(* Schneider Machine Expert - Basic project Project_M221_ModbusRTU_Master, file version 2.8.0.0 *)
(* ProjectInformations: Name=New project *)

HARDWARE
  Cpu 0: TM221ME16T/G
  ModuleExtensionObject 0: TM3SAF5R/G
  EthernetConfiguration: NetworkName=M221, IpAllocationMode=FixedAddress, IpAddress=192.168.5.84, SubnetMask=255.255.255.0
  SerialLineConfiguration: Baud=Baud115200, Parity=ParityEven, DataBits=DataBits8, StopBits=StopBits1, PhysicalMedium=PhysicalMediumRs485, TransmissionMode=TransmissionModeModbusRtu, SlaveId=1, Addressing=MasterAddressing
  MastTask: UsePeriodScanMode=true, PeriodScan=1
  FastTask: Period=255
  CpuBehavior: StartingMode=StartAsPreviousState, AutoSaveRamOnEeprom=true, WatchdogPeriod=250

SYMBOLS  (address, symbol, comment, settings)
  %M0       HMI_SW_ADD1
  %M1       HMI_SW_RESET
  %M2       HMI_LP_INSETPOINT
  %M10      READVAR_MODE03_EXEXUTE
  %M11      READVAR_MODE03_ABORT
  %M12      READVAR_MODE03_DONE
  %M13      READVAR_MODE03_BUSY
  %M14      READVAR_MODE03_ABORTED
  %M15      READVAR_MODE03_ERROR
  %M20      WRITEVAR_MODE10_EXECUTE
  %M21      WRITEVAR_MODE10_ABORT
  %M22      WRITEVAR_MODE10_DONE
  %M23      WRITEVAR_MODE10_BUSY
  %M24      WRITEVAR_MODE10_ABORTED
  %M25      WRITEVAR_MODE10_ERROR
  %M30      READVAR_MODE02_EXECUTE
  %M31      READVAR_MODE02_ABORT
  %M32      READVAR_MODE02_DONE
  %M33      READVAR_MODE02_BUSY
  %M34      READVAR_MODE02_ABORTED
  %M35      READVAR_MODE02_ERROR
  %M40      WRITEVAR_MODE0F_EXECUTE
  %M41      WRITEVAR_MODE0F_ABORT
  %M42      WRITEVAR_MODE0F_DONE
  %M43      WRITEVAR_MODE0F_BUSY
  %M44      WRITEVAR_MODE0F_ABORTED
  %M45      WRITEVAR_MODE0F_ERROR
  %M50      READVAR_MODE01_EXECUTE
  %M51      READVAR_MODE01_ABORT
  %M52      READVAR_MODE01_DONE
  %M53      READVAR_MODE01_BUSY
  %M54      READVAR_MODE01_ABORTED
  %M55      READVAR_MODE01_ERROR
  %M60      WRITEVAR_MODE06_EXECUTE
  %M61      WRITEVAR_MODE06_ABORT
  %M62      WRITEVAR_MODE06_DONE
  %M63      WRITEVAR_MODE06_BUSY
  %M64      WRITEVAR_MODE06_ABORTED
  %M65      WRITEVAR_MODE06_ERROR
  %M70      WRITEVAR_MODE05_EXECUTE
  %M71      WRITEVAR_MODE05_ABORT
  %M72      WRITEVAR_MODE05_DONE
  %M73      WRITEVAR_MODE05_BUSY
  %M74      WRITEVAR_MODE05_ABORTED
  %M75      WRITEVAR_MODE05_ERROR
  %M80      READVAR_MODE04_EXECUTE
  %M81      READVAR_MODE04_ABORT
  %M82      READVAR_MODE04_DONE
  %M83      READVAR_MODE04_BUSY
  %M84      READVAR_MODE04_ABORTED
  %M85      READVAR_MODE04_ERROR
  %M100       "VALID"
  %M101       "ERRORSTOP"
  %M102       "DISABLED"
  %M103       "STOPPING"
  %M104       "STANDSTILL"
  %M105       "CONTMOTION"
  %M106       "ERROR"
  %M107       "DONE"
  %M108       "BUSY"
  %M109       "ERROR"
  %M500     DUMMY
  %S12      SB_RUNMODE  "The controller is running"
  %MW0      RTU_REGISTER_0
  %MW1      ISTEP
  %MW2      RTU_REGISTER_2
  %MW3      OKCOUNT
  %MW4      RTU_REGISTER_4
  %MW5      RTU_REGISTER_5
  %MW6      RTU_REGISTER_6
  %MW7      RTU_REGISTER_7
  %MW8      RTU_REGISTER_8
  %MW9      RTU_REGISTER_9
  %MW10     RTU_REGISTER_10
  %MW11     RTU_REGISTER_11
  %MW12     RTU_REGISTER_12
  %MW13     RTU_REGISTER_13
  %MW14     RTU_REGISTER_14
  %MW100    MULTIREGISTER_0
  %MW101    MULTIREGISTER_1
  %MW102    MULTIREGISTER_2
  %MW400    READ_VAR1_BUFFER
  %MW402    WRITE_VAR1_BUFFER
  %MW404    READ_VAR2_BUFFER
  %MW410    READ_VAR0_BUFFER0
  %MW411    READ_VAR0_BUFFER1
  %MW412    READ_VAR0_BUFFER2
  %MW413    READ_VAR0_BUFFER3
  %MW414    READ_VAR0_BUFFER4
  %MW415    READ_VAR0_BUFFER5
  %MW416    READ_VAR0_BUFFER6
  %MW417    READ_VAR0_BUFFER7
  %MW418    READ_VAR0_BUFFER8
  %MW419    READ_VAR0_BUFFER9
  %MW420    READ_VAR3_BUFFER0
  %MW421    READ_VAR3_BUFFER1
  %MW422    READ_VAR3_BUFFER2
  %MW423    READ_VAR3_BUFFER3
  %MW424    READ_VAR3_BUFFER4
  %MW425    READ_VAR3_BUFFER5
  %MW426    READ_VAR3_BUFFER6
  %MW427    READ_VAR3_BUFFER7
  %MW428    READ_VAR3_BUFFER8
  %MW429    READ_VAR3_BUFFER9
  %MW430    WRITE_VAR0_BUFFER0
  %MW431    WRITE_VAR0_BUFFER1
  %MW432    WRITE_VAR0_BUFFER2
  %MW433    WRITE_VAR0_BUFFER3
  %MW434    WRITE_VAR0_BUFFER4
  %MW435    WRITE_VAR0_BUFFER5
  %MW436    WRITE_VAR0_BUFFER6
  %MW437    WRITE_VAR0_BUFFER7
  %MW438    WRITE_VAR0_BUFFER8
  %MW439    WRITE_VAR0_BUFFER9
  %MW440    WRITE_VAR2_BUFFER0
  %MW441    WRITE_VAR3_BUFFER0
  %READ_VAR0 RTU_ID1_READ400000_10  [Link(Value(FBComLinkParameterEnums=SerialLine1)), RemoteDeviceId(Value(int=1)), Timeout(Value(int=200)), ObjType(Value(FBComObjTypeParameterEnums=MW)), FirstObj(Value(int=0)), Quantity(Value(int=10)), IndexData(Value(int=410))]
  %READ_VAR1 RTU_ID1_READ000000_16  [Link(Value(FBComLinkParameterEnums=SerialLine1)), RemoteDeviceId(Value(int=1)), Timeout(Value(int=100)), ObjType(Value(FBComObjTypeParameterEnums=I)), FirstObj(Value(int=0)), Quantity(Value(int=16)), IndexData(Value(int=400))]
  %READ_VAR2 RTU_ID1_READ000001_16  [Link(Value(FBComLinkParameterEnums=SerialLine1)), RemoteDeviceId(Value(int=1)), Timeout(Value(int=100)), ObjType(Value(FBComObjTypeParameterEnums=Q)), FirstObj(Value(int=0)), Quantity(Value(int=16)), IndexData(Value(int=404))]
  %READ_VAR3 RTU_ID1_READ300000_10  [Link(Value(FBComLinkParameterEnums=SerialLine1)), RemoteDeviceId(Value(int=1)), Timeout(Value(int=100)), ObjType(Value(FBComObjTypeParameterEnums=IW)), FirstObj(Value(int=0)), Quantity(Value(int=10)), IndexData(Value(int=420))]
  %WRITE_VAR0 RTU_ID1_WRITE300000_10  [Link(Value(FBComLinkParameterEnums=SerialLine1)), RemoteDeviceId(Value(int=1)), Timeout(Value(int=100)), ObjType(Value(FBComObjTypeParameterEnums=MW)), FirstObj(Value(int=0)), Quantity(Value(int=10)), IndexData(Value(int=430))]
  %WRITE_VAR1 RTU_ID1_WRITE000000_16  [Link(Value(FBComLinkParameterEnums=SerialLine1)), RemoteDeviceId(Value(int=1)), Timeout(Value(int=100)), ObjType(Value(FBComObjTypeParameterEnums=Q)), FirstObj(Value(int=0)), Quantity(Value(int=16)), IndexData(Value(int=402))]
  %WRITE_VAR2 RTU_ID1_WRITE400000_1  [Link(Value(FBComLinkParameterEnums=SerialLine1)), RemoteDeviceId(Value(int=1)), Timeout(Value(int=100)), ObjType(Value(FBComObjTypeParameterEnums=SINGLE_REG)), FirstObj(Value(int=14)), Quantity(Value(int=1)), IndexData(Value(int=440))]
  %WRITE_VAR3 RTU_ID1_WRITE000000_1  [Link(Value(FBComLinkParameterEnums=SerialLine1)), RemoteDeviceId(Value(int=1)), Timeout(Value(int=100)), ObjType(Value(FBComObjTypeParameterEnums=SINGLE_COIL)), FirstObj(Value(int=0)), Quantity(Value(int=1)), IndexData(Value(int=441))]
  %QWM0     MODBUS_QWM0
  %QWM1     MODBUS_QWM1
  %QWM2     MODBUS_QWM2
  %QWM3     MODBUS_QWM3
  %QWM4     MODBUS_QWM4
  %QWM5     MODBUS_QWM5
  %QWM6     MODBUS_QWM6
  %QWM7     MODBUS_QWM7
  %QWM8     MODBUS_QWM8
  %QWM9     MODBUS_QWM9
  %QWM10    MODBUS_QWM10
  %QWM11    MODBUS_QWM11
  %QWM12    MODBUS_QWM12
  %QWM13    MODBUS_QWM13
  %QWM14    MODBUS_QWM14
  %QWM15    MODBUS_QWM15
  %QWM16    MODBUS_QWM16
  %QWM17    MODBUS_QWM17
  %QWM18    MODBUS_QWM18
  %QWM19    MODBUS_QWM19
  %IWM0     MODBUS_IWM0
  %IWM1     MODBUS_IWM1
  %IWM2     MODBUS_IWM2
  %IWM3     MODBUS_IWM3
  %IWM4     MODBUS_IWM4
  %IWM5     MODBUS_IWM5
  %IWM6     MODBUS_IWM6
  %IWM7     MODBUS_IWM7
  %IWM8     MODBUS_IWM8
  %IWM9     MODBUS_IWM9
  %IWM10    MODBUS_IWM10
  %IWM11    MODBUS_IWM11
  %IWM12    MODBUS_IWM12
  %IWM13    MODBUS_IWM13
  %IWM14    MODBUS_IWM14
  %IWM15    MODBUS_IWM15
  %IWM16    MODBUS_IWM16
  %IWM17    MODBUS_IWM17
  %IWM18    MODBUS_IWM18
  %IWM19    MODBUS_IWM19
  %I1.8       "Reserved"
  %I1.13      "Reserved"
  %Q1.3       "Reserved"

POU Pou01_System
  (* SectionNumber=1 *)

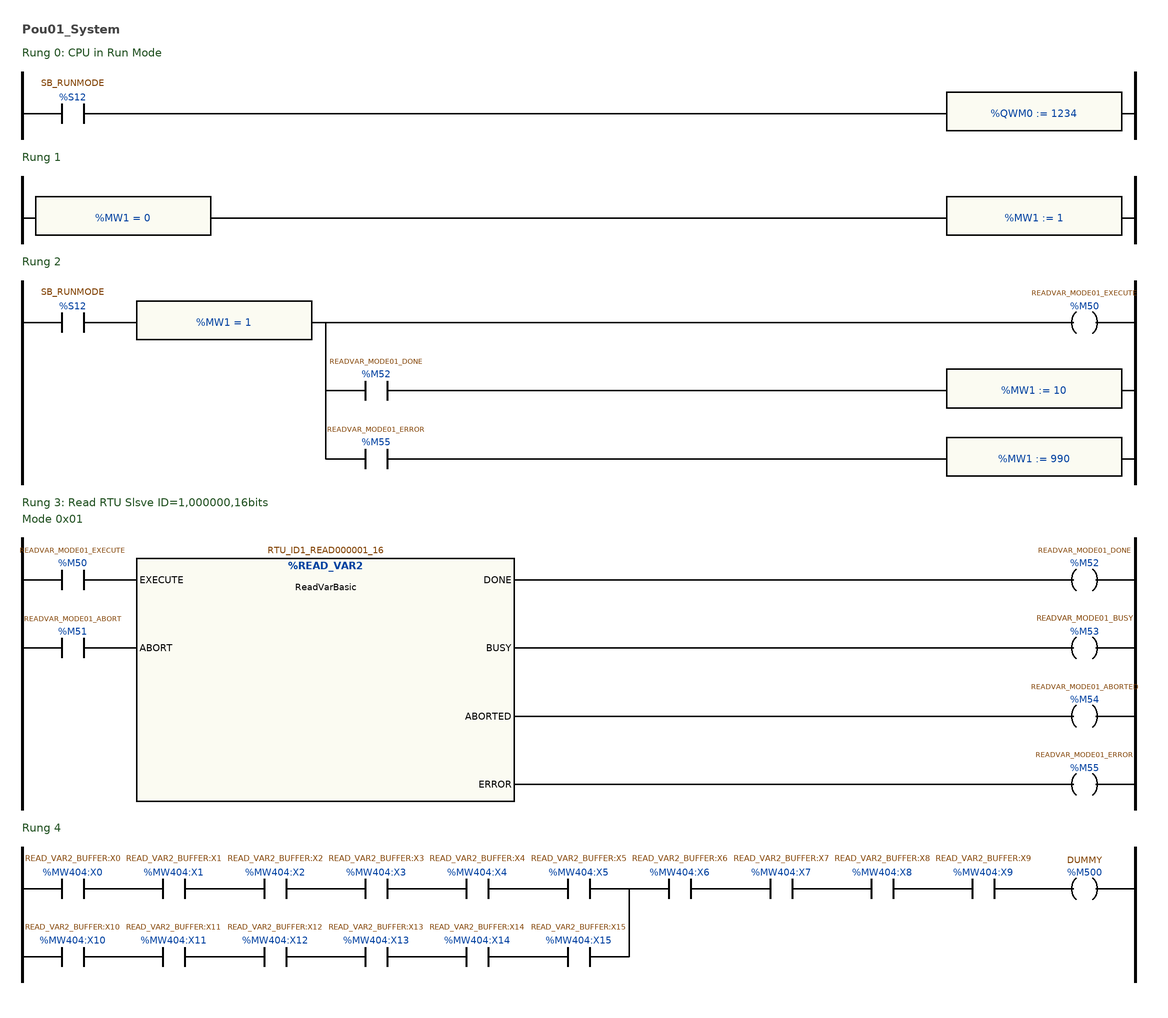

// Rung 0: CPU in Run Mode
  LD %S12                 (* SB_RUNMODE *)
  [ %QWM0 := 1234 ]       (* MODBUS_QWM0 *)
  // as ST:
  //   IF SB_RUNMODE THEN MODBUS_QWM0 := 1234; END_IF;

// Rung 1
  LD [ %MW1 = 0 ]         (* ISTEP *)
  [ %MW1 := 1 ]           (* ISTEP *)
  // as ST:
  //   IF ISTEP = 0 THEN ISTEP := 1; END_IF;

// Rung 2
  LD %S12                 (* SB_RUNMODE *)
  AND [ %MW1 = 1 ]        (* ISTEP *)
  MPS
  ST %M50                 (* READVAR_MODE01_EXECUTE *)
  MRD
  AND %M52                (* READVAR_MODE01_DONE *)
  [ %MW1 := 10 ]          (* ISTEP *)
  MPP
  AND %M55                (* READVAR_MODE01_ERROR *)
  [ %MW1 := 990 ]         (* ISTEP *)
  // as ST:
  //   READVAR_MODE01_EXECUTE := SB_RUNMODE AND ISTEP = 1;
  //   _t1 := SB_RUNMODE AND ISTEP = 1;
  //   IF SB_RUNMODE AND ISTEP = 1 AND READVAR_MODE01_DONE THEN ISTEP := 10; END_IF;
  //   IF _t1 AND READVAR_MODE01_ERROR THEN ISTEP := 990; END_IF;

// Rung 3: Read RTU Slsve ID=1,000000,16bits
// Mode 0x01
  BLK %READ_VAR2
  LD %M50                 (* READVAR_MODE01_EXECUTE *)
  EXECUTE
  LD %M51                 (* READVAR_MODE01_ABORT *)
  ABORT
  OUT_BLK
  LD DONE
  ST %M52                 (* READVAR_MODE01_DONE *)
  LD BUSY
  ST %M53                 (* READVAR_MODE01_BUSY *)
  LD ABORTED
  ST %M54                 (* READVAR_MODE01_ABORTED *)
  LD ERROR
  ST %M55                 (* READVAR_MODE01_ERROR *)
  END_BLK
  // as ST:
  //   %READ_VAR2(EXECUTE := READVAR_MODE01_EXECUTE, ABORT := READVAR_MODE01_ABORT);
  //   READVAR_MODE01_DONE := %READ_VAR2.DONE;
  //   READVAR_MODE01_BUSY := %READ_VAR2.BUSY;
  //   READVAR_MODE01_ABORTED := %READ_VAR2.ABORTED;
  //   READVAR_MODE01_ERROR := %READ_VAR2.ERROR;

// Rung 4
  LD %MW404:X0            (* READ_VAR2_BUFFER *)
  AND %MW404:X1           (* READ_VAR2_BUFFER *)
  AND %MW404:X2           (* READ_VAR2_BUFFER *)
  AND %MW404:X3           (* READ_VAR2_BUFFER *)
  AND %MW404:X4           (* READ_VAR2_BUFFER *)
  AND %MW404:X5           (* READ_VAR2_BUFFER *)
  OR( %MW404:X10          (* READ_VAR2_BUFFER *)
  AND %MW404:X11          (* READ_VAR2_BUFFER *)
  AND %MW404:X12          (* READ_VAR2_BUFFER *)
  AND %MW404:X13          (* READ_VAR2_BUFFER *)
  AND %MW404:X14          (* READ_VAR2_BUFFER *)
  AND %MW404:X15          (* READ_VAR2_BUFFER *)
  )
  AND %MW404:X6           (* READ_VAR2_BUFFER *)
  AND %MW404:X7           (* READ_VAR2_BUFFER *)
  AND %MW404:X8           (* READ_VAR2_BUFFER *)
  AND %MW404:X9           (* READ_VAR2_BUFFER *)
  ST %M500                (* DUMMY *)
  // as ST:
  //   DUMMY := (READ_VAR2_BUFFER:X0 AND READ_VAR2_BUFFER:X1 AND READ_VAR2_BUFFER:X2 AND READ_VAR2_BUFFER:X3 AND READ_VAR2_BUFFER:X4 AND READ_VAR2_BUFFER:X5 OR READ_VAR2_BUFFER:X10 AND READ_VAR2_BUFFER:X11 AND READ_VAR2_BUFFER:X12 AND READ_VAR2_BUFFER:X13 AND READ_VAR2_BUFFER:X14 AND READ_VAR2_BUFFER:X15) AND READ_VAR2_BUFFER:X6 AND READ_VAR2_BUFFER:X7 AND READ_VAR2_BUFFER:X8 AND READ_VAR2_BUFFER:X9;

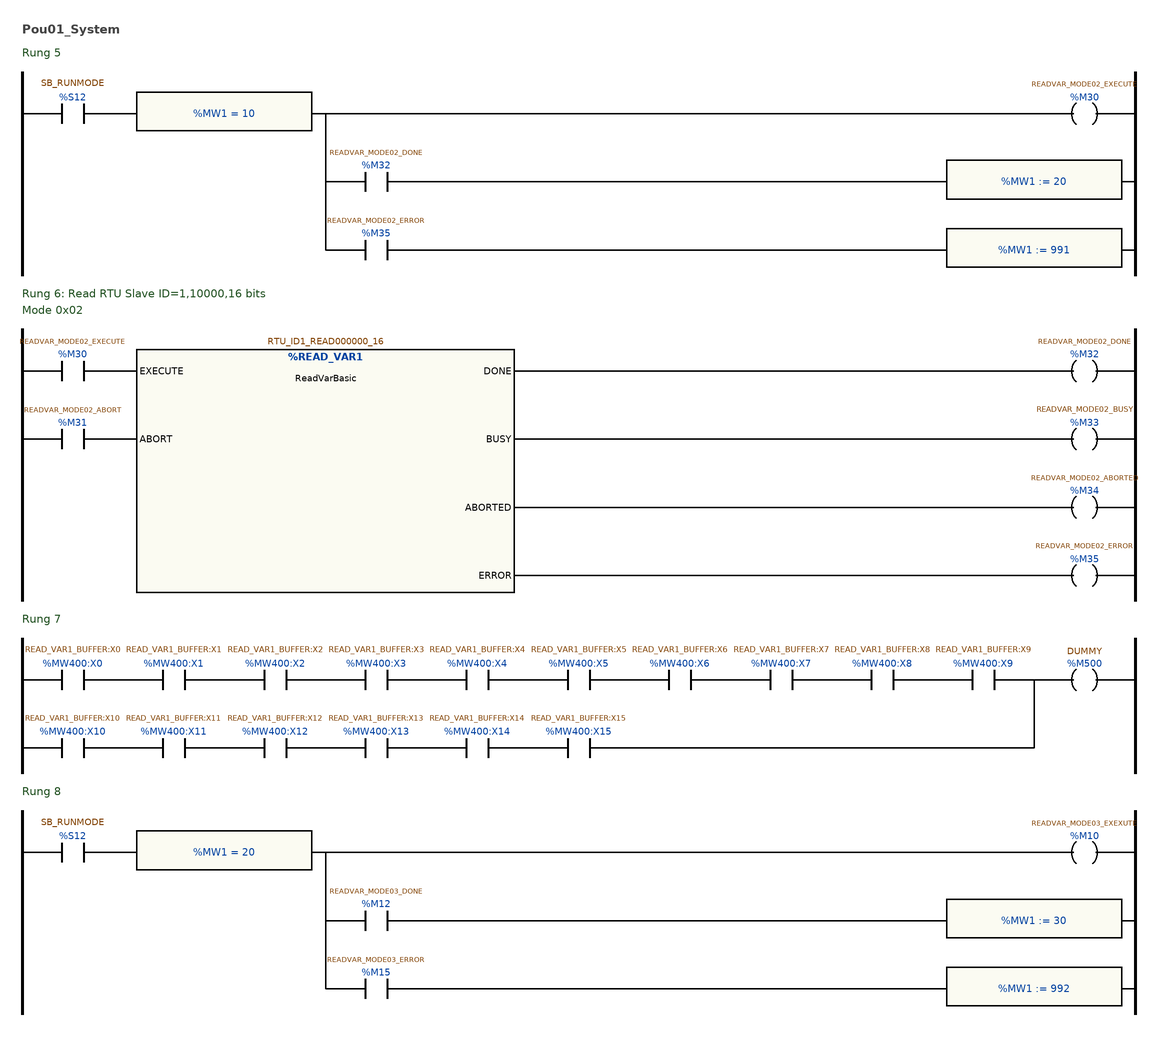

// Rung 5
  LD %S12                 (* SB_RUNMODE *)
  AND [ %MW1 = 10 ]       (* ISTEP *)
  MPS
  ST %M30                 (* READVAR_MODE02_EXECUTE *)
  MRD
  AND %M32                (* READVAR_MODE02_DONE *)
  [ %MW1 := 20 ]          (* ISTEP *)
  MPP
  AND %M35                (* READVAR_MODE02_ERROR *)
  [ %MW1 := 991 ]         (* ISTEP *)
  // as ST:
  //   READVAR_MODE02_EXECUTE := SB_RUNMODE AND ISTEP = 10;
  //   _t1 := SB_RUNMODE AND ISTEP = 10;
  //   IF SB_RUNMODE AND ISTEP = 10 AND READVAR_MODE02_DONE THEN ISTEP := 20; END_IF;
  //   IF _t1 AND READVAR_MODE02_ERROR THEN ISTEP := 991; END_IF;

// Rung 6: Read RTU Slave ID=1,10000,16 bits
// Mode 0x02
  BLK %READ_VAR1
  LD %M30                 (* READVAR_MODE02_EXECUTE *)
  EXECUTE
  LD %M31                 (* READVAR_MODE02_ABORT *)
  ABORT
  OUT_BLK
  LD DONE
  ST %M32                 (* READVAR_MODE02_DONE *)
  LD BUSY
  ST %M33                 (* READVAR_MODE02_BUSY *)
  LD ABORTED
  ST %M34                 (* READVAR_MODE02_ABORTED *)
  LD ERROR
  ST %M35                 (* READVAR_MODE02_ERROR *)
  END_BLK
  // as ST:
  //   %READ_VAR1(EXECUTE := READVAR_MODE02_EXECUTE, ABORT := READVAR_MODE02_ABORT);
  //   READVAR_MODE02_DONE := %READ_VAR1.DONE;
  //   READVAR_MODE02_BUSY := %READ_VAR1.BUSY;
  //   READVAR_MODE02_ABORTED := %READ_VAR1.ABORTED;
  //   READVAR_MODE02_ERROR := %READ_VAR1.ERROR;

// Rung 7
  LD %MW400:X0            (* READ_VAR1_BUFFER *)
  AND %MW400:X1           (* READ_VAR1_BUFFER *)
  AND %MW400:X2           (* READ_VAR1_BUFFER *)
  AND %MW400:X3           (* READ_VAR1_BUFFER *)
  AND %MW400:X4           (* READ_VAR1_BUFFER *)
  AND %MW400:X5           (* READ_VAR1_BUFFER *)
  AND %MW400:X6           (* READ_VAR1_BUFFER *)
  AND %MW400:X7           (* READ_VAR1_BUFFER *)
  AND %MW400:X8           (* READ_VAR1_BUFFER *)
  AND %MW400:X9           (* READ_VAR1_BUFFER *)
  OR( %MW400:X10          (* READ_VAR1_BUFFER *)
  AND %MW400:X11          (* READ_VAR1_BUFFER *)
  AND %MW400:X12          (* READ_VAR1_BUFFER *)
  AND %MW400:X13          (* READ_VAR1_BUFFER *)
  AND %MW400:X14          (* READ_VAR1_BUFFER *)
  AND %MW400:X15          (* READ_VAR1_BUFFER *)
  )
  ST %M500                (* DUMMY *)
  // as ST:
  //   DUMMY := READ_VAR1_BUFFER:X0 AND READ_VAR1_BUFFER:X1 AND READ_VAR1_BUFFER:X2 AND READ_VAR1_BUFFER:X3 AND READ_VAR1_BUFFER:X4 AND READ_VAR1_BUFFER:X5 AND READ_VAR1_BUFFER:X6 AND READ_VAR1_BUFFER:X7 AND READ_VAR1_BUFFER:X8 AND READ_VAR1_BUFFER:X9 OR READ_VAR1_BUFFER:X10 AND READ_VAR1_BUFFER:X11 AND READ_VAR1_BUFFER:X12 AND READ_VAR1_BUFFER:X13 AND READ_VAR1_BUFFER:X14 AND READ_VAR1_BUFFER:X15;

// Rung 8
  LD %S12                 (* SB_RUNMODE *)
  AND [ %MW1 = 20 ]       (* ISTEP *)
  MPS
  ST %M10                 (* READVAR_MODE03_EXEXUTE *)
  MRD
  AND %M12                (* READVAR_MODE03_DONE *)
  [ %MW1 := 30 ]          (* ISTEP *)
  MPP
  AND %M15                (* READVAR_MODE03_ERROR *)
  [ %MW1 := 992 ]         (* ISTEP *)
  // as ST:
  //   READVAR_MODE03_EXEXUTE := SB_RUNMODE AND ISTEP = 20;
  //   _t1 := SB_RUNMODE AND ISTEP = 20;
  //   IF SB_RUNMODE AND ISTEP = 20 AND READVAR_MODE03_DONE THEN ISTEP := 30; END_IF;
  //   IF _t1 AND READVAR_MODE03_ERROR THEN ISTEP := 992; END_IF;

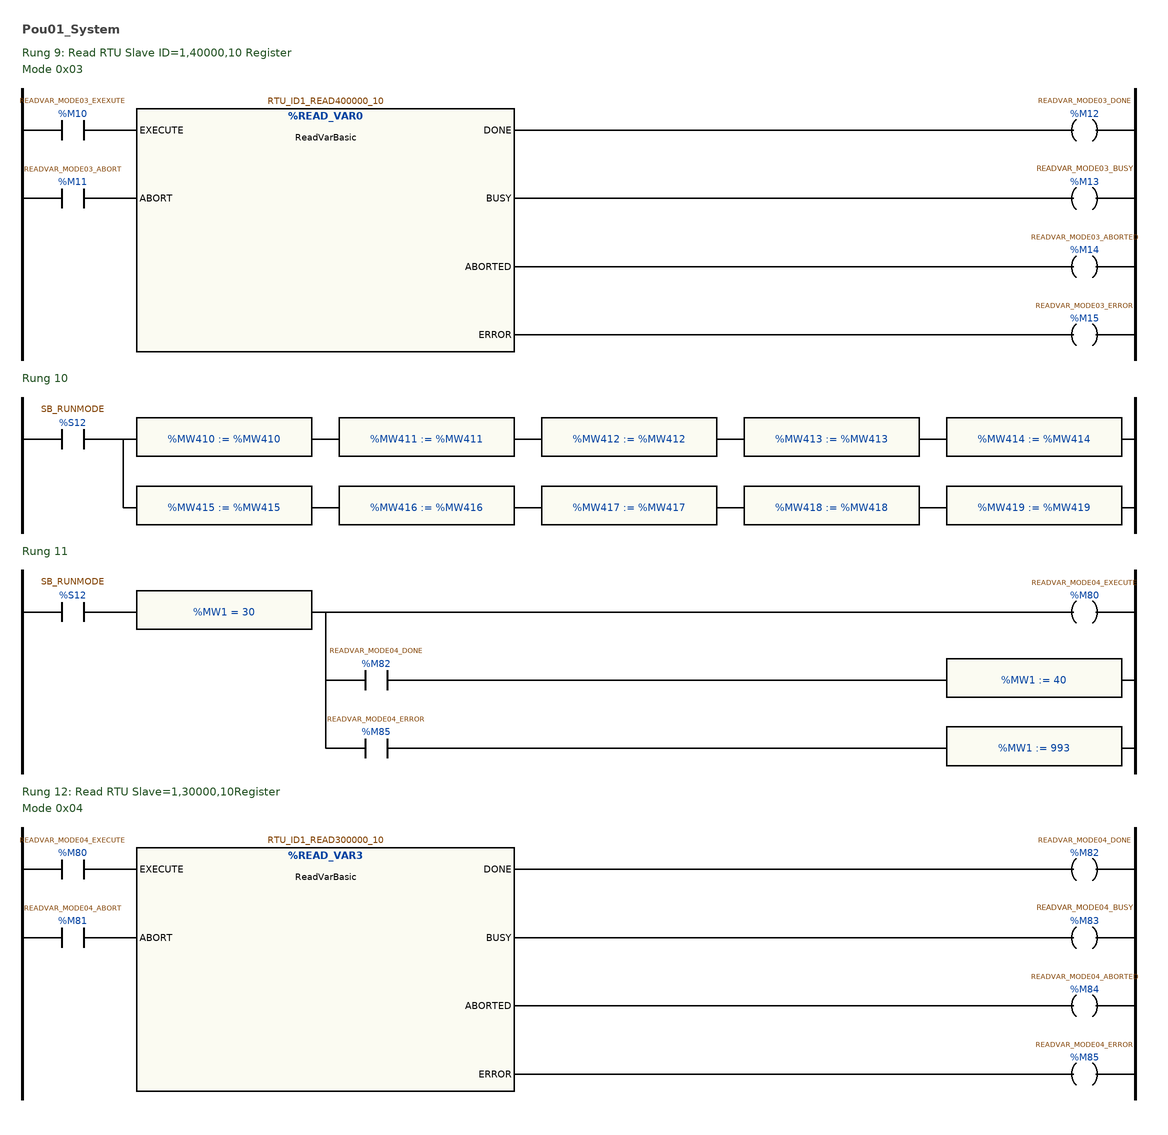

// Rung 9: Read RTU Slave ID=1,40000,10 Register
// Mode 0x03
  BLK %READ_VAR0
  LD %M10                 (* READVAR_MODE03_EXEXUTE *)
  EXECUTE
  LD %M11                 (* READVAR_MODE03_ABORT *)
  ABORT
  OUT_BLK
  LD DONE
  ST %M12                 (* READVAR_MODE03_DONE *)
  LD BUSY
  ST %M13                 (* READVAR_MODE03_BUSY *)
  LD ABORTED
  ST %M14                 (* READVAR_MODE03_ABORTED *)
  LD ERROR
  ST %M15                 (* READVAR_MODE03_ERROR *)
  END_BLK
  // as ST:
  //   %READ_VAR0(EXECUTE := READVAR_MODE03_EXEXUTE, ABORT := READVAR_MODE03_ABORT);
  //   READVAR_MODE03_DONE := %READ_VAR0.DONE;
  //   READVAR_MODE03_BUSY := %READ_VAR0.BUSY;
  //   READVAR_MODE03_ABORTED := %READ_VAR0.ABORTED;
  //   READVAR_MODE03_ERROR := %READ_VAR0.ERROR;

// Rung 10
  LD %S12                 (* SB_RUNMODE *)
  MPS
  OPER [ %MW410 := %MW410 ](* READ_VAR0_BUFFER0, READ_VAR0_BUFFER0 *)
  OPER [ %MW411 := %MW411 ](* READ_VAR0_BUFFER1, READ_VAR0_BUFFER1 *)
  OPER [ %MW412 := %MW412 ](* READ_VAR0_BUFFER2, READ_VAR0_BUFFER2 *)
  OPER [ %MW413 := %MW413 ](* READ_VAR0_BUFFER3, READ_VAR0_BUFFER3 *)
  [ %MW414 := %MW414 ]    (* READ_VAR0_BUFFER4, READ_VAR0_BUFFER4 *)
  MPP
  OPER [ %MW415 := %MW415 ](* READ_VAR0_BUFFER5, READ_VAR0_BUFFER5 *)
  OPER [ %MW416 := %MW416 ](* READ_VAR0_BUFFER6, READ_VAR0_BUFFER6 *)
  OPER [ %MW417 := %MW417 ](* READ_VAR0_BUFFER7, READ_VAR0_BUFFER7 *)
  OPER [ %MW418 := %MW418 ](* READ_VAR0_BUFFER8, READ_VAR0_BUFFER8 *)
  [ %MW419 := %MW419 ]    (* READ_VAR0_BUFFER9, READ_VAR0_BUFFER9 *)
  // as ST:
  //   IF SB_RUNMODE THEN READ_VAR0_BUFFER0 := READ_VAR0_BUFFER0; END_IF;
  //   IF SB_RUNMODE THEN READ_VAR0_BUFFER1 := READ_VAR0_BUFFER1; END_IF;
  //   IF SB_RUNMODE THEN READ_VAR0_BUFFER2 := READ_VAR0_BUFFER2; END_IF;
  //   IF SB_RUNMODE THEN READ_VAR0_BUFFER3 := READ_VAR0_BUFFER3; END_IF;
  //   IF SB_RUNMODE THEN READ_VAR0_BUFFER4 := READ_VAR0_BUFFER4; END_IF;
  //   IF SB_RUNMODE THEN READ_VAR0_BUFFER5 := READ_VAR0_BUFFER5; END_IF;
  //   IF SB_RUNMODE THEN READ_VAR0_BUFFER6 := READ_VAR0_BUFFER6; END_IF;
  //   IF SB_RUNMODE THEN READ_VAR0_BUFFER7 := READ_VAR0_BUFFER7; END_IF;
  //   IF SB_RUNMODE THEN READ_VAR0_BUFFER8 := READ_VAR0_BUFFER8; END_IF;
  //   IF SB_RUNMODE THEN READ_VAR0_BUFFER9 := READ_VAR0_BUFFER9; END_IF;

// Rung 11
  LD %S12                 (* SB_RUNMODE *)
  AND [ %MW1 = 30 ]       (* ISTEP *)
  MPS
  ST %M80                 (* READVAR_MODE04_EXECUTE *)
  MRD
  AND %M82                (* READVAR_MODE04_DONE *)
  [ %MW1 := 40 ]          (* ISTEP *)
  MPP
  AND %M85                (* READVAR_MODE04_ERROR *)
  [ %MW1 := 993 ]         (* ISTEP *)
  // as ST:
  //   READVAR_MODE04_EXECUTE := SB_RUNMODE AND ISTEP = 30;
  //   _t1 := SB_RUNMODE AND ISTEP = 30;
  //   IF SB_RUNMODE AND ISTEP = 30 AND READVAR_MODE04_DONE THEN ISTEP := 40; END_IF;
  //   IF _t1 AND READVAR_MODE04_ERROR THEN ISTEP := 993; END_IF;

// Rung 12: Read RTU Slave=1,30000,10Register
// Mode 0x04
  BLK %READ_VAR3
  LD %M80                 (* READVAR_MODE04_EXECUTE *)
  EXECUTE
  LD %M81                 (* READVAR_MODE04_ABORT *)
  ABORT
  OUT_BLK
  LD DONE
  ST %M82                 (* READVAR_MODE04_DONE *)
  LD BUSY
  ST %M83                 (* READVAR_MODE04_BUSY *)
  LD ABORTED
  ST %M84                 (* READVAR_MODE04_ABORTED *)
  LD ERROR
  ST %M85                 (* READVAR_MODE04_ERROR *)
  END_BLK
  // as ST:
  //   %READ_VAR3(EXECUTE := READVAR_MODE04_EXECUTE, ABORT := READVAR_MODE04_ABORT);
  //   READVAR_MODE04_DONE := %READ_VAR3.DONE;
  //   READVAR_MODE04_BUSY := %READ_VAR3.BUSY;
  //   READVAR_MODE04_ABORTED := %READ_VAR3.ABORTED;
  //   READVAR_MODE04_ERROR := %READ_VAR3.ERROR;

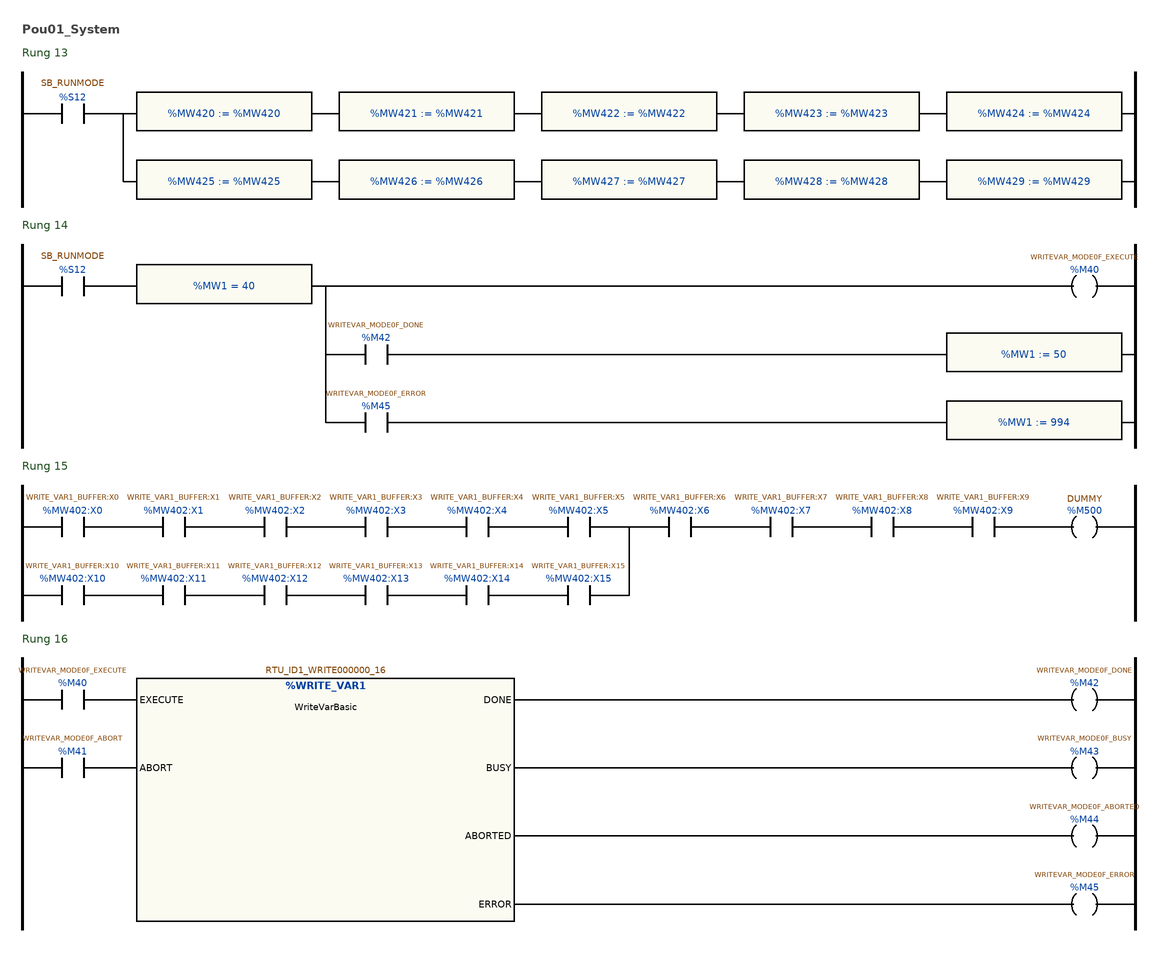

// Rung 13
  LD %S12                 (* SB_RUNMODE *)
  MPS
  OPER [ %MW420 := %MW420 ](* READ_VAR3_BUFFER0, READ_VAR3_BUFFER0 *)
  OPER [ %MW421 := %MW421 ](* READ_VAR3_BUFFER1, READ_VAR3_BUFFER1 *)
  OPER [ %MW422 := %MW422 ](* READ_VAR3_BUFFER2, READ_VAR3_BUFFER2 *)
  OPER [ %MW423 := %MW423 ](* READ_VAR3_BUFFER3, READ_VAR3_BUFFER3 *)
  [ %MW424 := %MW424 ]    (* READ_VAR3_BUFFER4, READ_VAR3_BUFFER4 *)
  MPP
  OPER [ %MW425 := %MW425 ](* READ_VAR3_BUFFER5, READ_VAR3_BUFFER5 *)
  OPER [ %MW426 := %MW426 ](* READ_VAR3_BUFFER6, READ_VAR3_BUFFER6 *)
  OPER [ %MW427 := %MW427 ](* READ_VAR3_BUFFER7, READ_VAR3_BUFFER7 *)
  OPER [ %MW428 := %MW428 ](* READ_VAR3_BUFFER8, READ_VAR3_BUFFER8 *)
  [ %MW429 := %MW429 ]    (* READ_VAR3_BUFFER9, READ_VAR3_BUFFER9 *)
  // as ST:
  //   IF SB_RUNMODE THEN READ_VAR3_BUFFER0 := READ_VAR3_BUFFER0; END_IF;
  //   IF SB_RUNMODE THEN READ_VAR3_BUFFER1 := READ_VAR3_BUFFER1; END_IF;
  //   IF SB_RUNMODE THEN READ_VAR3_BUFFER2 := READ_VAR3_BUFFER2; END_IF;
  //   IF SB_RUNMODE THEN READ_VAR3_BUFFER3 := READ_VAR3_BUFFER3; END_IF;
  //   IF SB_RUNMODE THEN READ_VAR3_BUFFER4 := READ_VAR3_BUFFER4; END_IF;
  //   IF SB_RUNMODE THEN READ_VAR3_BUFFER5 := READ_VAR3_BUFFER5; END_IF;
  //   IF SB_RUNMODE THEN READ_VAR3_BUFFER6 := READ_VAR3_BUFFER6; END_IF;
  //   IF SB_RUNMODE THEN READ_VAR3_BUFFER7 := READ_VAR3_BUFFER7; END_IF;
  //   IF SB_RUNMODE THEN READ_VAR3_BUFFER8 := READ_VAR3_BUFFER8; END_IF;
  //   IF SB_RUNMODE THEN READ_VAR3_BUFFER9 := READ_VAR3_BUFFER9; END_IF;

// Rung 14
  LD %S12                 (* SB_RUNMODE *)
  AND [ %MW1 = 40 ]       (* ISTEP *)
  MPS
  ST %M40                 (* WRITEVAR_MODE0F_EXECUTE *)
  MRD
  AND %M42                (* WRITEVAR_MODE0F_DONE *)
  [ %MW1 := 50 ]          (* ISTEP *)
  MPP
  AND %M45                (* WRITEVAR_MODE0F_ERROR *)
  [ %MW1 := 994 ]         (* ISTEP *)
  // as ST:
  //   WRITEVAR_MODE0F_EXECUTE := SB_RUNMODE AND ISTEP = 40;
  //   _t1 := SB_RUNMODE AND ISTEP = 40;
  //   IF SB_RUNMODE AND ISTEP = 40 AND WRITEVAR_MODE0F_DONE THEN ISTEP := 50; END_IF;
  //   IF _t1 AND WRITEVAR_MODE0F_ERROR THEN ISTEP := 994; END_IF;

// Rung 15
  LD %MW402:X0            (* WRITE_VAR1_BUFFER *)
  AND %MW402:X1           (* WRITE_VAR1_BUFFER *)
  AND %MW402:X2           (* WRITE_VAR1_BUFFER *)
  AND %MW402:X3           (* WRITE_VAR1_BUFFER *)
  AND %MW402:X4           (* WRITE_VAR1_BUFFER *)
  AND %MW402:X5           (* WRITE_VAR1_BUFFER *)
  OR( %MW402:X10          (* WRITE_VAR1_BUFFER *)
  AND %MW402:X11          (* WRITE_VAR1_BUFFER *)
  AND %MW402:X12          (* WRITE_VAR1_BUFFER *)
  AND %MW402:X13          (* WRITE_VAR1_BUFFER *)
  AND %MW402:X14          (* WRITE_VAR1_BUFFER *)
  AND %MW402:X15          (* WRITE_VAR1_BUFFER *)
  )
  AND %MW402:X6           (* WRITE_VAR1_BUFFER *)
  AND %MW402:X7           (* WRITE_VAR1_BUFFER *)
  AND %MW402:X8           (* WRITE_VAR1_BUFFER *)
  AND %MW402:X9           (* WRITE_VAR1_BUFFER *)
  ST %M500                (* DUMMY *)
  // as ST:
  //   DUMMY := (WRITE_VAR1_BUFFER:X0 AND WRITE_VAR1_BUFFER:X1 AND WRITE_VAR1_BUFFER:X2 AND WRITE_VAR1_BUFFER:X3 AND WRITE_VAR1_BUFFER:X4 AND WRITE_VAR1_BUFFER:X5 OR WRITE_VAR1_BUFFER:X10 AND WRITE_VAR1_BUFFER:X11 AND WRITE_VAR1_BUFFER:X12 AND WRITE_VAR1_BUFFER:X13 AND WRITE_VAR1_BUFFER:X14 AND WRITE_VAR1_BUFFER:X15) AND WRITE_VAR1_BUFFER:X6 AND WRITE_VAR1_BUFFER:X7 AND WRITE_VAR1_BUFFER:X8 AND WRITE_VAR1_BUFFER:X9;

// Rung 16
  BLK %WRITE_VAR1
  LD %M40                 (* WRITEVAR_MODE0F_EXECUTE *)
  EXECUTE
  LD %M41                 (* WRITEVAR_MODE0F_ABORT *)
  ABORT
  OUT_BLK
  LD DONE
  ST %M42                 (* WRITEVAR_MODE0F_DONE *)
  LD BUSY
  ST %M43                 (* WRITEVAR_MODE0F_BUSY *)
  LD ABORTED
  ST %M44                 (* WRITEVAR_MODE0F_ABORTED *)
  LD ERROR
  ST %M45                 (* WRITEVAR_MODE0F_ERROR *)
  END_BLK
  // as ST:
  //   %WRITE_VAR1(EXECUTE := WRITEVAR_MODE0F_EXECUTE, ABORT := WRITEVAR_MODE0F_ABORT);
  //   WRITEVAR_MODE0F_DONE := %WRITE_VAR1.DONE;
  //   WRITEVAR_MODE0F_BUSY := %WRITE_VAR1.BUSY;
  //   WRITEVAR_MODE0F_ABORTED := %WRITE_VAR1.ABORTED;
  //   WRITEVAR_MODE0F_ERROR := %WRITE_VAR1.ERROR;

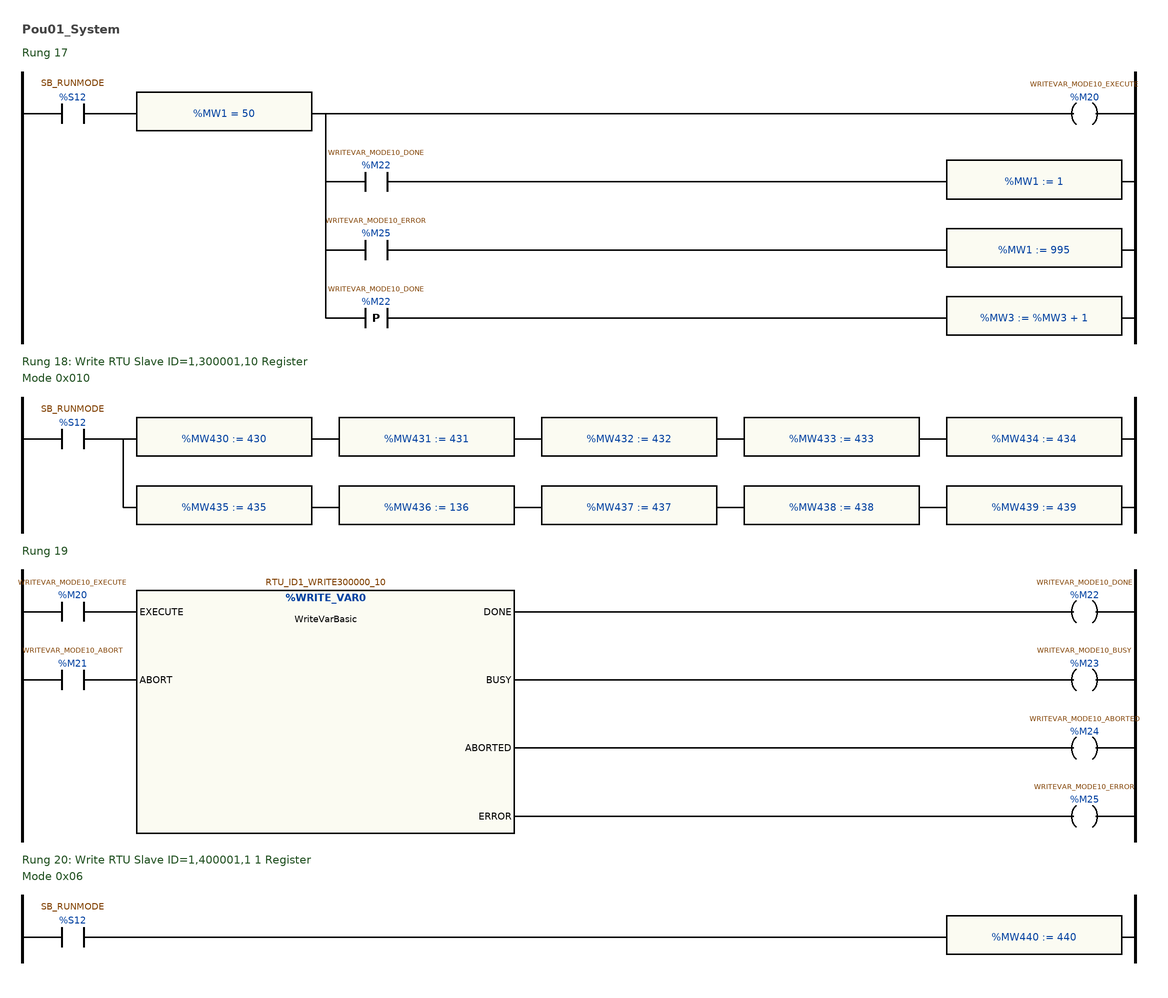

// Rung 17
  LD %S12                 (* SB_RUNMODE *)
  AND [ %MW1 = 50 ]       (* ISTEP *)
  MPS
  ST %M20                 (* WRITEVAR_MODE10_EXECUTE *)
  MRD
  AND %M22                (* WRITEVAR_MODE10_DONE *)
  [ %MW1 := 1 ]           (* ISTEP *)
  MRD
  AND %M25                (* WRITEVAR_MODE10_ERROR *)
  [ %MW1 := 995 ]         (* ISTEP *)
  MPP
  ANDR %M22               (* WRITEVAR_MODE10_DONE *)
  [ %MW3 := %MW3 + 1 ]    (* OKCOUNT, OKCOUNT *)
  // as ST:
  //   WRITEVAR_MODE10_EXECUTE := SB_RUNMODE AND ISTEP = 50;
  //   _t1 := SB_RUNMODE AND ISTEP = 50;
  //   IF SB_RUNMODE AND ISTEP = 50 AND WRITEVAR_MODE10_DONE THEN ISTEP := 1; END_IF;
  //   IF _t1 AND WRITEVAR_MODE10_ERROR THEN ISTEP := 995; END_IF;
  //   IF _t1 AND RISING(WRITEVAR_MODE10_DONE) THEN OKCOUNT := OKCOUNT + 1; END_IF;

// Rung 18: Write RTU Slave ID=1,300001,10 Register
// Mode 0x010
  LD %S12                 (* SB_RUNMODE *)
  MPS
  OPER [ %MW430 := 430 ]  (* WRITE_VAR0_BUFFER0 *)
  OPER [ %MW431 := 431 ]  (* WRITE_VAR0_BUFFER1 *)
  OPER [ %MW432 := 432 ]  (* WRITE_VAR0_BUFFER2 *)
  OPER [ %MW433 := 433 ]  (* WRITE_VAR0_BUFFER3 *)
  [ %MW434 := 434 ]       (* WRITE_VAR0_BUFFER4 *)
  MPP
  OPER [ %MW435 := 435 ]  (* WRITE_VAR0_BUFFER5 *)
  OPER [ %MW436 := 136 ]  (* WRITE_VAR0_BUFFER6 *)
  OPER [ %MW437 := 437 ]  (* WRITE_VAR0_BUFFER7 *)
  OPER [ %MW438 := 438 ]  (* WRITE_VAR0_BUFFER8 *)
  [ %MW439 := 439 ]       (* WRITE_VAR0_BUFFER9 *)
  // as ST:
  //   IF SB_RUNMODE THEN WRITE_VAR0_BUFFER0 := 430; END_IF;
  //   IF SB_RUNMODE THEN WRITE_VAR0_BUFFER1 := 431; END_IF;
  //   IF SB_RUNMODE THEN WRITE_VAR0_BUFFER2 := 432; END_IF;
  //   IF SB_RUNMODE THEN WRITE_VAR0_BUFFER3 := 433; END_IF;
  //   IF SB_RUNMODE THEN WRITE_VAR0_BUFFER4 := 434; END_IF;
  //   IF SB_RUNMODE THEN WRITE_VAR0_BUFFER5 := 435; END_IF;
  //   IF SB_RUNMODE THEN WRITE_VAR0_BUFFER6 := 136; END_IF;
  //   IF SB_RUNMODE THEN WRITE_VAR0_BUFFER7 := 437; END_IF;
  //   IF SB_RUNMODE THEN WRITE_VAR0_BUFFER8 := 438; END_IF;
  //   IF SB_RUNMODE THEN WRITE_VAR0_BUFFER9 := 439; END_IF;

// Rung 19
  BLK %WRITE_VAR0
  LD %M20                 (* WRITEVAR_MODE10_EXECUTE *)
  EXECUTE
  LD %M21                 (* WRITEVAR_MODE10_ABORT *)
  ABORT
  OUT_BLK
  LD DONE
  ST %M22                 (* WRITEVAR_MODE10_DONE *)
  LD BUSY
  ST %M23                 (* WRITEVAR_MODE10_BUSY *)
  LD ABORTED
  ST %M24                 (* WRITEVAR_MODE10_ABORTED *)
  LD ERROR
  ST %M25                 (* WRITEVAR_MODE10_ERROR *)
  END_BLK
  // as ST:
  //   %WRITE_VAR0(EXECUTE := WRITEVAR_MODE10_EXECUTE, ABORT := WRITEVAR_MODE10_ABORT);
  //   WRITEVAR_MODE10_DONE := %WRITE_VAR0.DONE;
  //   WRITEVAR_MODE10_BUSY := %WRITE_VAR0.BUSY;
  //   WRITEVAR_MODE10_ABORTED := %WRITE_VAR0.ABORTED;
  //   WRITEVAR_MODE10_ERROR := %WRITE_VAR0.ERROR;

// Rung 20: Write RTU Slave ID=1,400001,1 1 Register
// Mode 0x06
  LD %S12                 (* SB_RUNMODE *)
  [ %MW440 := 440 ]       (* WRITE_VAR2_BUFFER0 *)
  // as ST:
  //   IF SB_RUNMODE THEN WRITE_VAR2_BUFFER0 := 440; END_IF;

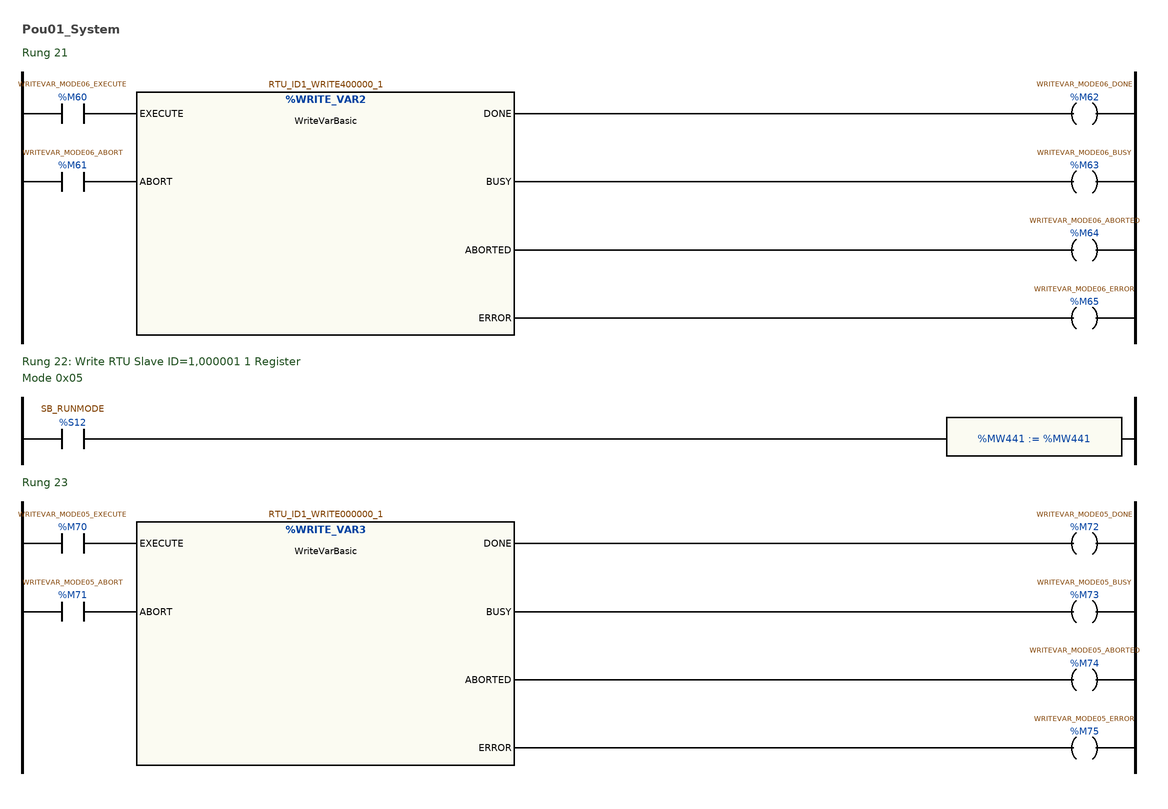

// Rung 21
  BLK %WRITE_VAR2
  LD %M60                 (* WRITEVAR_MODE06_EXECUTE *)
  EXECUTE
  LD %M61                 (* WRITEVAR_MODE06_ABORT *)
  ABORT
  OUT_BLK
  LD DONE
  ST %M62                 (* WRITEVAR_MODE06_DONE *)
  LD BUSY
  ST %M63                 (* WRITEVAR_MODE06_BUSY *)
  LD ABORTED
  ST %M64                 (* WRITEVAR_MODE06_ABORTED *)
  LD ERROR
  ST %M65                 (* WRITEVAR_MODE06_ERROR *)
  END_BLK
  // as ST:
  //   %WRITE_VAR2(EXECUTE := WRITEVAR_MODE06_EXECUTE, ABORT := WRITEVAR_MODE06_ABORT);
  //   WRITEVAR_MODE06_DONE := %WRITE_VAR2.DONE;
  //   WRITEVAR_MODE06_BUSY := %WRITE_VAR2.BUSY;
  //   WRITEVAR_MODE06_ABORTED := %WRITE_VAR2.ABORTED;
  //   WRITEVAR_MODE06_ERROR := %WRITE_VAR2.ERROR;

// Rung 22: Write RTU Slave ID=1,000001 1 Register
// Mode 0x05
  LD %S12                 (* SB_RUNMODE *)
  [ %MW441 := %MW441 ]    (* WRITE_VAR3_BUFFER0, WRITE_VAR3_BUFFER0 *)
  // as ST:
  //   IF SB_RUNMODE THEN WRITE_VAR3_BUFFER0 := WRITE_VAR3_BUFFER0; END_IF;

// Rung 23
  BLK %WRITE_VAR3
  LD %M70                 (* WRITEVAR_MODE05_EXECUTE *)
  EXECUTE
  LD %M71                 (* WRITEVAR_MODE05_ABORT *)
  ABORT
  OUT_BLK
  LD DONE
  ST %M72                 (* WRITEVAR_MODE05_DONE *)
  LD BUSY
  ST %M73                 (* WRITEVAR_MODE05_BUSY *)
  LD ABORTED
  ST %M74                 (* WRITEVAR_MODE05_ABORTED *)
  LD ERROR
  ST %M75                 (* WRITEVAR_MODE05_ERROR *)
  END_BLK
  // as ST:
  //   %WRITE_VAR3(EXECUTE := WRITEVAR_MODE05_EXECUTE, ABORT := WRITEVAR_MODE05_ABORT);
  //   WRITEVAR_MODE05_DONE := %WRITE_VAR3.DONE;
  //   WRITEVAR_MODE05_BUSY := %WRITE_VAR3.BUSY;
  //   WRITEVAR_MODE05_ABORTED := %WRITE_VAR3.ABORTED;
  //   WRITEVAR_MODE05_ERROR := %WRITE_VAR3.ERROR;
